{attribute 'qualified_only'}
VAR_GLOBAL
	AL_1 AT %I* : INT;
	AL_2 AT %I* : INT;
	AL_3 AT %I* : INT;
	AL_4 AT %I* : INT;
END_VAR

(* stored: Version 1.1.0.1
   GVL ANALOG: Id {848e0958-298c-4369-9d58-493c584afcb3} *)
